// TwinCAT 3 PLC project PLC1
// ProgramVersion: 3.1.4026.15
// libraries:
//   Tc2_Standard, * (Beckhoff Automation GmbH)
//   Tc2_System, * (Beckhoff Automation GmbH)
//   Tc2_Utilities, * (Beckhoff Automation GmbH)
// project tree:
//   / PlcTask.TcTTO
//   SYS/DUTs/ E_OperatingMode.TcDUT, E_SystemState.TcDUT, ST_Part.TcDUT, ST_SA.TcDUT, ST_TypeSt.TcDUT, ST_TypeTr.TcDUT
//   SYS/FBs/Mode/ FB_ConsoleLogger.TcPOU, FB_ModeStateMachine.TcPOU, FB_SA.TcPOU, FB_ZoneControl.TcPOU
//   SYS/FBs/Sim/ FB_SIM.TcPOU
//   SYS/FBs/Time/ FB_GetTime.TcPOU, FB_Time.TcPOU
//   SYS/FBs/Type/ FB_TypeControl.TcPOU, FB_TypeShift.TcPOU
//   SYS/FCs/ generatePartID.TcPOU
//   SYS/GVLs/ GLOB.TcGVL, SIM.TcGVL
//   SYS/IF/ IEventLogger.TcIO
//   SYS/ MAIN.TcPOU
//   USER/Cfg/ Cfg.TcPOU
//   USER/ STU_Part.TcDUT, U.TcGVL, U_MAIN.TcPOU
//   USER/Type Shifting/ U_Typeshift.TcPOU
// real-time tasks:
//   TASK PlcTask: cycle T#10ms, priority 20, ADS port 350

CONFIGURATION PLC1
    RESOURCE PLC ON TwinCAT3
        TASK PlcTask(INTERVAL := T#10ms, PRIORITY := 20);
        PROGRAM MAIN WITH PlcTask : MAIN;
    END_RESOURCE
END_CONFIGURATION

// ---- SYS/DUTs/E_OperatingMode.TcDUT
{attribute 'qualified_only'}
{attribute 'strict'}
{attribute 'to_string'}
TYPE E_OperatingMode :
(
    eMode_Manual := 0,
    eMode_Auto   := 1,
    eMode_Error  := 2
);
END_TYPE

// ---- SYS/DUTs/E_SystemState.TcDUT
{attribute 'qualified_only'}
{attribute 'strict'}
{attribute 'to_string'}
TYPE E_SystemState  :
(
    eState_Init := 0,
    eState_Manual,
    eState_AutoIdle,
	eState_AutoRunning,
	eState_Error
);
END_TYPE

// ---- SYS/DUTs/ST_Part.TcDUT
TYPE ST_Part :
STRUCT
	runningNumber	: INT;
	variant			: INT;
	ID				: STRING;
	timeStamp		: INT;
	route			: INT;
	scrap			: BOOL;
	jobs			: DINT;
	user			: STU_Part;
END_STRUCT
END_TYPE

// ---- SYS/DUTs/ST_SA.TcDUT
TYPE ST_SA :
STRUCT
	name		: STRING;
	ID			: INT;
	EstopOK		: BOOL;
	GatesOK		: BOOL;
	SafetyOK	: BOOL;
END_STRUCT
END_TYPE

// ---- SYS/DUTs/ST_TypeSt.TcDUT
TYPE ST_TypeSt :
STRUCT
	name		: STRING;
	part		: ST_Part;
	withPart	: BOOL;
	nextType	: BOOL;
	jobDone		: BOOL;
	hold		: BOOL;
	noWork		: BOOL;
	inPos1		: BOOL;
	inPos2		: BOOL;
	processTime	: REAL;
	designTime	: REAL	:= 5;
	nextSt		: INT;
END_STRUCT
END_TYPE

// ---- SYS/DUTs/ST_TypeTr.TcDUT
TYPE ST_TypeTr :
STRUCT
	fromSt		: INT;
	toSt		: INT;
	enabled		: INT;
	part		: ST_Part;
	withPart	: BOOL;
	nextType	: BOOL;
	jobDone		: BOOL;
	hold		: BOOL;
	noWork		: BOOL;
	inPos1		: BOOL;
	inPos2		: BOOL;
	processTime	: REAL;
	designTime	: REAL	:= 3;
	nextSt		: INT;
END_STRUCT
END_TYPE

// ---- USER/STU_Part.TcDUT
TYPE STU_Part :
STRUCT
	user1	: BOOL;
	user2	: BOOL;
	user3	: INT;
	user4	: INT;	
END_STRUCT
END_TYPE

// ---- SYS/GVLs/GLOB.TcGVL
{attribute 'qualified_only'}
VAR_GLOBAL
	bStart		: BOOL;
	bStop		: BOOL;
	bReset		: BOOL;
	bAuto		: BOOL;
	bManual		: BOOL;
	bFault		: BOOL;
	bSelectAll	: BOOL;
	RNR			: INT;
	bShuttle	: BOOL;
	partID		: STRING;
END_VAR

// ---- SYS/GVLs/SIM.TcGVL
{attribute 'qualified_only'}
VAR_GLOBAL
	active		: BOOL;
	generate	: BOOL;
	shift		: BOOL;
	delete		: BOOL;
	safetyNOK	: BOOL;
	fault		: BOOL;
END_VAR

// ---- USER/U.TcGVL
//{attribute 'qualified_only'}
VAR_GLOBAL CONSTANT
	MAX_SA_NR	: INT	:= 10;
	MAX_ST_NR	: INT	:= 30;
	MAX_VAR_NR	: INT	:= 9;
	
END_VAR
VAR_GLOBAL
	SA			: ARRAY [0..MAX_SA_NR] OF ST_SA;	
	typeSt		: ARRAY [0..MAX_ST_NR] OF ST_TypeSt;
	typeTr		: ARRAY [0..MAX_ST_NR] OF ST_TypeTr;
END_VAR

// ---- SYS/IF/IEventLogger.TcIO
INTERFACE IEventLogger

METHOD LogEvent : bool
VAR_INPUT
	sMessage : STRING;
END_VAR
END_METHOD

END_INTERFACE

// ---- SYS/MAIN.TcPOU
PROGRAM MAIN
VAR
	Simulation		: FB_SIM;
	TypeControl		: FB_TypeControl;
	TypeUser		: U_Typeshift;
	Zone1			: FB_ZoneControl;
	Zone2			: FB_ZoneControl;
	Zone3			: FB_ZoneControl;	
	GenFault		: BOOL;
	userMain		: U_Main;	
	timing			: FB_Time;
	
	bInitDone		: BOOL;
	nCounter		: ULINT;
END_VAR

// Init
IF NOT bInitDone THEN
    // Init Settings
	Zone1.sZoneName := 'Zone A';
	Zone2.sZoneName := 'Zone B';
	Zone3.sZoneName := 'Zone X';
    bInitDone := TRUE;
END_IF


// Calls
timing();
Simulation();
userMain();
TypeControl();
Zone1(bError := Glob.bFault);
Zone2(bError := Glob.bFault);
Zone3(bError := Glob.bFault);


// Running Counter
nCounter	:=	nCounter + 1;

END_PROGRAM

// ---- SYS/FBs/Sim/FB_SIM.TcPOU
FUNCTION_BLOCK FB_SIM
VAR_INPUT
END_VAR
VAR_OUTPUT
END_VAR
VAR
	generateEnable	: BOOL;
	shiftEnable		: BOOL;
	index			: INT;
	variant			: INT;
	
END_VAR

// SIM JOB
IF SIM.active THEN
	FOR index := 1 TO MAX_ST_NR DO
		IF typeSt[index].processTime >= typeSt[index].designTime THEN
			typeSt[index].jobDone := TRUE;
		END_IF
	END_FOR
END_IF

// SIM PART
variant	:= variant + 1;
IF variant > MAX_VAR_NR THEN
	variant := 1;
END_IF
generateEnable	:= NOT typeSt[1].withPart;
IF generateEnable AND SIM.generate THEN
	GLOB.RNR	:= GLOB.RNR + 1;
	typeSt[1].part.runningNumber := GLOB.RNR;
	typeSt[1].part.variant	:= variant;
	typeSt[1].part.ID		:= GLOB.partID;
	typeSt[1].withPart	:= TRUE;	
END_IF

// SIM SHIFT
shiftEnable 	:= typeSt[1].jobDone AND NOT typeSt[2].withPart;
IF shiftEnable AND SIM.shift THEN
	typeSt[2].part	:= typeSt[1].part;
	typeSt[1].part	:= typeSt[0].part;
	//MEMSET(destAddr:= typeSt[1].part, fillByte:= 0, n:= 1);
	typeSt[2].withPart := TRUE;
	typeSt[1].withPart := FALSE;		
END_IF

END_FUNCTION_BLOCK

// ---- SYS/FBs/Type/FB_TypeControl.TcPOU
FUNCTION_BLOCK FB_TypeControl
VAR_INPUT
END_VAR
VAR_OUTPUT
END_VAR
VAR
	initDone	: BOOL;
	index	: INT;
	//typeSt010	: REFERENCE OF typeSt[1];
END_VAR

// TYPE LOOP
FOR index := 1 TO MAX_ST_NR DO
	IF typeSt[index].withPart THEN 
		typeSt[index].nextType := FALSE;
		typeSt[index].processTime := typeSt[index].processTime + 0.01;
	ELSE
		typeSt[index].processTime	:= 0;
		typeSt[index].jobDone := FALSE;
		typeSt[index].part	:= typeSt[0].part;
	END_IF	
END_FOR

END_FUNCTION_BLOCK

// ---- USER/Type Shifting/U_Typeshift.TcPOU
FUNCTION_BLOCK U_Typeshift
VAR_INPUT
END_VAR
VAR_OUTPUT
END_VAR
VAR
	Shift01_02		: FB_TypeShift;
	Shift02_03		: FB_TypeShift;
	Shift02_04		: FB_TypeShift;
	Shift03_05		: FB_TypeShift;
	Shift04_05		: FB_TypeShift;	
	Shift05_06		: FB_TypeShift;
	Shift06_07		: FB_TypeShift;	
	Shift07_08		: FB_TypeShift;
	Shift08_09		: FB_TypeShift;
	Shift08_16		: FB_TypeShift;
	Shift09_10		: FB_TypeShift;
	Shift10_11		: FB_TypeShift;
	Shift11_12		: FB_TypeShift;
	Shift12_13		: FB_TypeShift;
	Shift13_14		: FB_TypeShift;
	Shift14_15		: FB_TypeShift;
	Shift15_01		: FB_TypeShift;
	Shift16_08		: FB_TypeShift;
END_VAR

// TYPE SHIFTING
Shift01_02(fromSt:= 1, toSt:= 2);
Shift02_03(fromSt:= 2, toSt:= 3);
Shift02_04(fromSt:= 2, toSt:= 4);
Shift03_05(fromSt:= 3, toSt:= 5);
Shift04_05(fromSt:= 4, toSt:= 5);
Shift05_06(fromSt:= 5, toSt:= 6);
Shift06_07(fromSt:= 6, toSt:= 7);
// insert part back to line prio to normal flow
IF NOT typeSt[16].part.scrap THEN
	Shift16_08(fromSt:= 16, toSt:= 08);
END_IF
Shift07_08(fromSt:= 7, toSt:= 8);
// extract part from line if scrap or continue
IF NOT typeSt[8].part.scrap THEN
	Shift08_09(fromSt:= 8, toSt:= 9);
END_IF
Shift08_16(fromSt:= 08, toSt:= 16,);
Shift09_10(fromSt:= 09, toSt:= 10,);
Shift10_11(fromSt:= 10, toSt:= 11);
Shift11_12(fromSt:= 11, toSt:= 12);
Shift12_13(fromSt:= 12, toSt:= 13);
Shift13_14(fromSt:= 13, toSt:= 14);
Shift14_15(fromSt:= 14, toSt:= 15);
Shift15_01(fromSt:= 15, toSt:= 01);

END_FUNCTION_BLOCK

// ---- SYS/FBs/Type/FB_TypeShift.TcPOU
FUNCTION_BLOCK FB_TypeShift
VAR_INPUT
	index			: INT;
	fromSt			: INT;
	toSt			: INT;
	shuttleAllowed	: BOOL;
END_VAR
VAR_OUTPUT
END_VAR
VAR
	enabled			: BOOL;
	shiftDelay		: TON;
END_VAR

//enabled := NOT typeTr[index].withPart AND NOT typeSt[toSt].withPart AND typeSt[fromSt].jobDone;
enabled :=	NOT typeSt[toSt].withPart
			AND typeSt[fromSt].withPart 
			AND typeSt[fromSt].jobDone 
			AND NOT typeSt[fromSt].hold;

shiftDelay(IN:= enabled, PT:= T#500MS);

IF shiftDelay.Q THEN
	typeSt[toSt].part	:= typeSt[fromSt].part;
	typeSt[fromSt].part	:= typeSt[0].part;
	//MEMSET(destAddr:= typeSt[1].part, fillByte:= 0, n:= 1);
	typeSt[toSt].withPart := TRUE;
	typeSt[FromSt].withPart := FALSE;	
END_IF

END_FUNCTION_BLOCK

// ---- SYS/FBs/Mode/FB_ZoneControl.TcPOU
FUNCTION_BLOCK FB_ZoneControl
VAR_INPUT
	sZoneName 		: STRING := 'ZoneXXX'; // Default name
    bAutoMode     	: BOOL; // true = request auto
    bManualMode   	: BOOL; // true = request manual
    bStart        	: BOOL;
    bStop         	: BOOL;
    bReset        	: BOOL;
	bError			: BOOL;
	bSelected		: BOOL;
END_VAR

VAR_OUTPUT
    eMode         : E_OperatingMode;
    sStatus       : STRING(255); // for faceplate display
END_VAR

VAR
    fbLogger          : FB_ConsoleLogger;
    fbStateMachine    : FB_ModeStateMachine;
    bInitDone         : BOOL := FALSE;
END_VAR

IF NOT bInitDone THEN
    fbStateMachine.SetLogger(fbLogger); // Inject logger
	fbStateMachine.sSourceName := sZoneName;
    bInitDone := TRUE;
END_IF

// Global select all zones
IF glob.bSelectAll THEN
	bSelected 	:= TRUE;
END_IF

// Connect buttons to state machine inputs
fbStateMachine.bManualReq 	:= bManualMode 	OR (bSelected AND GLOB.bManual);
fbStateMachine.bAutoReq   	:= bAutoMode 	OR (bSelected AND GLOB.bauto);
fbStateMachine.bStart		:= bStart		OR (bSelected AND GLOB.bStart);
fbStateMachine.bStop		:= bStop		OR (bSelected AND GLOB.bStop);
fbStateMachine.bReset		:= bReset		OR (bSelected AND GLOB.bReset);
fbStateMachine.bError     	:= bError; 

// Run logic
fbStateMachine.Run();

// Update outputs
eMode   := fbStateMachine.eCurrentMode;
//sStatus := fbLogger.sLastMessage; // Optional — could show most recent log
sStatus := TO_STRING(fbStateMachine.estate);

END_FUNCTION_BLOCK

// ---- SYS/FBs/Mode/FB_ConsoleLogger.TcPOU
FUNCTION_BLOCK FB_ConsoleLogger IMPLEMENTS IEventLogger
VAR_INPUT
END_VAR
VAR_OUTPUT
	 sLastMessage : STRING(255);
END_VAR
VAR
END_VAR

{analysis 'TcLog'}
METHOD LogEvent : BOOL
VAR_INPUT
	sMessage	: STRING;
END_VAR
sLastMessage := sMessage;
LogEvent := TRUE; 

ADSLOGSTR(msgCtrlMask:= ADSLOG_MSGTYPE_HINT, msgFmtStr:= 'My log message: %s', strArg:= sMessage);
END_METHOD

END_FUNCTION_BLOCK

// ---- SYS/FBs/Mode/FB_ModeStateMachine.TcPOU
FUNCTION_BLOCK FB_ModeStateMachine
VAR_INPUT
	sSourceName 	: STRING := 'Unnamed';
    bManualReq 		: BOOL;
    bAutoReq   		: BOOL;
	bStart			: BOOL;
	bStop			: BOOL;
	bReset			: BOOL;
    bError     		: BOOL;
END_VAR

VAR_OUTPUT
    eCurrentMode : E_OperatingMode;
END_VAR

VAR
    eState       			: E_SystemState := E_SystemState.eState_Init;
    prevState   			: E_SystemState := E_SystemState.eState_Init;
    ePreviousNonErrorState 	: E_SystemState := E_SystemState.eState_Manual;
    logger       : IEventLogger; // Dependency injection
END_VAR

METHOD Run
VAR_INPUT
END_VAR
prevState := eState;

CASE eState OF

    E_SystemState.eState_Init:
        eCurrentMode := E_OperatingMode.eMode_Manual;
        eState := E_SystemState.eState_Manual;

    E_SystemState.eState_Manual:
        eCurrentMode := E_OperatingMode.eMode_Manual;
        IF bAutoReq THEN
            eState := E_SystemState.eState_AutoIdle;
        ELSIF bError THEN
			ePreviousNonErrorState := eState;
			eState := E_SystemState.eState_Error;
        END_IF

	E_SystemState.eState_AutoIdle:
	    eCurrentMode := E_OperatingMode.eMode_Auto;
	
	    IF bStart THEN
	        eState := E_SystemState.eState_AutoRunning;
	    ELSIF bManualReq THEN
	        eState := E_SystemState.eState_Manual;
	    ELSIF bError THEN
			ePreviousNonErrorState := eState;
	        eState := E_SystemState.eState_Error;
	    END_IF
	
	E_SystemState.eState_AutoRunning:
	    eCurrentMode := E_OperatingMode.eMode_Auto;
	
	    IF bStop THEN
	        eState := E_SystemState.eState_AutoIdle;
	    ELSIF bManualReq THEN
	        eState := E_SystemState.eState_Manual;
	    ELSIF bError THEN
			ePreviousNonErrorState := eState;
	        eState := E_SystemState.eState_Error;
	    END_IF

	E_SystemState.eState_Error:
	    eCurrentMode := E_OperatingMode.eMode_Error;
	
	    IF bReset AND NOT bError THEN
	        CASE ePreviousNonErrorState OF
	            E_SystemState.eState_Manual:
	                eState := E_SystemState.eState_Manual;
	
	            E_SystemState.eState_AutoIdle,
	            E_SystemState.eState_AutoRunning:
	                eState := E_SystemState.eState_AutoIdle;
	
	            ELSE
	                eState := E_SystemState.eState_Manual;
	        END_CASE
	    END_IF


END_CASE

IF eState <> prevState THEN
    logger.LogEvent(sMessage := CONCAT(CONCAT(sSourceName, ' - Transitioned to: '), TO_STRING(eState)));
END_IF
END_METHOD

METHOD SetLogger
VAR_INPUT
	fbLogger : IEventLogger;
END_VAR
logger	:= fbLogger;
END_METHOD

END_FUNCTION_BLOCK

// ---- USER/U_MAIN.TcPOU
FUNCTION_BLOCK U_MAIN
VAR_INPUT
END_VAR
VAR_OUTPUT
END_VAR
VAR
	initDone	: BOOL;
	typeshift	: U_typeshift;
END_VAR

IF NOT initDone THEN
	Cfg();
	initDone := TRUE;	
END_IF

//calls
typeshift();

END_FUNCTION_BLOCK

// ---- USER/Cfg/Cfg.TcPOU
FUNCTION Cfg
VAR_INPUT
END_VAR
VAR
END_VAR

// Naming Safety Area's
SA[1].name	:= 'SA01';

// Naming Type Station and Design Time
typeSt[1].name := 'ST010';
typeSt[1].designTime := 3;
typeSt[2].name := 'ST020';
typeSt[3].name := 'ST030 (PRIM)';
typeSt[3].designTime := 10;
typeSt[4].name := 'ST035 (SEC)';
typeSt[4].designTime := 10;
typeSt[5].name := 'ST040';
typeSt[6].name := 'ST050';
typeSt[7].name := 'ST060';
typeSt[8].name := 'ST070';
typeSt[9].name := 'ST080';
typeSt[10].name := 'ST090';
typeSt[11].name := 'ST100';
typeSt[12].name := 'ST115';
typeSt[13].name := 'ST120';
typeSt[14].name := 'ST130';
typeSt[15].name := 'ST140';
typeSt[16].name := 'REPAIR';

END_FUNCTION

// ---- SYS/FBs/Time/FB_Time.TcPOU
FUNCTION_BLOCK FB_Time
VAR_INPUT
END_VAR
VAR_OUTPUT
END_VAR
VAR
	runOnce				: BOOL	:= TRUE;
	timeCall			: FB_GetTime;
	systemTime			: ULINT;
	timeAsStruct		: TIMESTRUCT;
	speed				: UINT := 1;
END_VAR

IF runOnce THEN
	runOnce := FALSE;
	systemTime := F_GetSystemTime();
END_IF

//systemTime := F_GetSystemTime();
systemTime		:= (systemTime + (speed * 100000)); 
timeAsStruct	:= FILETIME64_TO_SYSTEMTIME(systemTime);


timeCall();
GLOB.partID	:= generatePartID(timeCall.isTime);

END_FUNCTION_BLOCK

// ---- SYS/FBs/Time/FB_GetTime.TcPOU
FUNCTION_BLOCK FB_GetTime
VAR_INPUT
END_VAR
VAR_OUTPUT
	isTime			: TIMESTRUCT;
END_VAR
VAR
	ticks			: ULINT;
	last			: ULINT;
	start			: BOOL;	
	getTime			: NT_GetTime;
END_VAR

ticks := ticks + 1;

start := FALSE;
IF ticks - last > 100 THEN
	last := ticks;
	start := TRUE;
END_IF
start := start AND NOT getTime.BUSY;

getTime(
	NETID:= , 
	START:= start, 
	TMOUT:= , 
	BUSY=> , 
	ERR=> , 
	ERRID=> , 
	TIMESTR=> isTime);

END_FUNCTION_BLOCK

// ---- SYS/FCs/generatePartID.TcPOU
FUNCTION generatePartID : STRING
VAR_INPUT
	timeStruct	: TIMESTRUCT;
END_VAR
VAR
	tempString	: STRING;
	monthString : STRING;
	dayString	: STRING;
	hourString	: STRING;
	minuteString: STRING;
	secondString: STRING;	
END_VAR

tempString	:= CONCAT('0', TO_STRING(timestruct.wMonth));
monthString := RIGHT(tempString,2);
tempString	:= CONCAT('0', TO_STRING(timestruct.wDay));
dayString 	:= RIGHT(tempString,2);
tempString	:= CONCAT('0', TO_STRING(timestruct.wHour));
hourString 	:= RIGHT(tempString,2);
tempString	:= CONCAT('0', TO_STRING(timestruct.wMinute));
minuteString:= RIGHT(tempString,2);
tempString	:= CONCAT('0', TO_STRING(timestruct.wSecond));
secondString:= RIGHT(tempString,2);

tempString	:= CONCAT(monthString, dayString);
tempString   := CONCAT(tempString, '-');
tempString	:= CONCAT(tempString, hourString);
tempString	:= CONCAT(tempString, minuteString);
tempString	:= CONCAT(tempString, secondString);

generatePartID:= tempString;

END_FUNCTION

// ---- SYS/FBs/Mode/FB_SA.TcPOU
FUNCTION_BLOCK FB_SA
VAR_INPUT
END_VAR
VAR_OUTPUT
END_VAR
VAR
END_VAR

END_FUNCTION_BLOCK
